// TIA Portal V16 export
// export: Created 2021-04-11T09:51:25.9267202Z, ExportSetting WithDefaults, DisplayName Totally Integrated Automation Portal, DisplayVersion V16, DisplayName TIA Portal Version Control Interface, DisplayVersion V16, DisplayName TIA Portal Openness, DisplayVersion V16, DisplayName STEP 7 Professional, DisplayVersion V16, DisplayName STEP 7 Safety, DisplayVersion V16, DisplayName WinCC Unified SCADA Engineering System, DisplayVersion V16
FUNCTION "set%Conv" : Void   // FC4, LAD
{ S7_Optimized_Access := 'TRUE' }
VERSION : 0.1
// stored: AutoNumber true, IsIECCheckEnabled false, SetENOAutomatically false, UDAEnableTagReadback false
   VAR_INPUT
      inPercent : Real;
      normMin : Real;
      normMax : Real;
      scaleMin : Real;
      scaleMax : Real;
   END_VAR
   VAR_OUTPUT
      bitValue : Int;
   END_VAR
   VAR_TEMP
      temp : Real;
   END_VAR
BEGIN

REGION Network 1
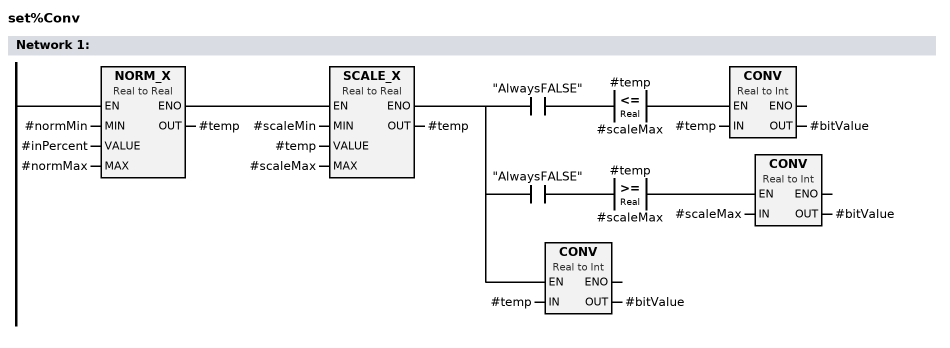
   RUNG wire#powerrail
      { S7_Templates := "[SrcType := Real, DestType := Real]" } Normalize(min := #normMin, value := #inPercent, max := #normMax, out => #temp)
      { S7_Templates := "[SrcType := Real, DestType := Real]" } Scale(min := #scaleMin, value := #temp, max := #scaleMax, out => #temp)
      wire#w1
      Contact( "AlwaysFALSE" )
      { S7_Templates := "SrcType := Real" } LE_Contact(in1 := #temp, in2 := #scaleMax)
      { S7_Templates := "[SrcType := Real, DestType := Int]" } Convert(in := #temp, out => #bitValue)
   END_RUNG
   RUNG wire#w1
      Contact( "AlwaysFALSE" )
      { S7_Templates := "SrcType := Real" } GE_Contact(in1 := #temp, in2 := #scaleMax)
      { S7_Templates := "[SrcType := Real, DestType := Int]" } Convert(in := #scaleMax, out => #bitValue)
   END_RUNG
   RUNG wire#w1
      { S7_Templates := "[SrcType := Real, DestType := Int]" } Convert(in := #temp, out => #bitValue)
   END_RUNG
   // the same network as SCL:
   #temp := NORM_X(MIN := #normMin, VALUE := #inPercent, MAX := #normMax);
   #temp := SCALE_X(MIN := #scaleMin, VALUE := #temp, MAX := #scaleMax);
   IF "AlwaysFALSE" AND (#temp <= #scaleMax) THEN #bitValue := REAL_TO_INT(#temp); END_IF;
   IF "AlwaysFALSE" AND (#temp >= #scaleMax) THEN #bitValue := REAL_TO_INT(#scaleMax); END_IF;
   #bitValue := REAL_TO_INT(#temp);
END_REGION
END_FUNCTION
